(* PLC project mainPLC, Beckhoff Automation GmbH TwinCAT PLC Control 3.5.13.21 *)
(* stored: creationDateTime 2022-08-21T13:19:37.4859706, modificationDateTime 2022-08-21T13:19:37.487966 *)

PROGRAM MAIN
VAR	
	PosDegree AT %I*	: REAL	:= 0;		// in deg
	PosPiston AT %I*	: REAL	:= 0;		// in mm
	velocity AT %Q*		: REAL	:= 0;		// in deg/s
	
	cycleTime 			: REAL := 0.01;		// in sec
END_VAR

            // Position of Disc
PosDegree := PosDegree + velocity*cycleTime;
WHILE PosDegree > 360 DO
	PosDegree := PosDegree -360;
END_WHILE


// Position of Piston    
PosPiston := 13 + COS(PosDegree*pi/180)*9 + SQRT(EXPT(25,2)-EXPT((SIN(PosDegree*pi/180 )*9),2));


          
END_PROGRAM
